FUNCTION_BLOCK fbEthercatStateMachine
VAR
	InputState AT%I*	:UINT;	
	WcState AT%I* :BOOL;
	InternalEtherCatState : st_EthercatState;
	
{attribute 'OPC.UA.DA' := '0'}	
	State :UINT;
		
{attribute 'OPC.UA.DA' := '0'}
	Error:UINT;
	
END_VAR

// table of states https://infosys.beckhoff.com/english.php?content=../content/1033/b110_ethercat_optioninterface/1984417163.html&id=
// uint is 16 bit final 4 bit are state first 12 are error 
State := InputState AND 16#000F;
Error := InputState AND 16#FFF0;
InternalEtherCatState.State:= UINT_TO_INT(State);
InternalEtherCatState.Error := UINT_TO_INT(Error);
InternalEtherCatState.DataInvalid := WcState;

METHOD FB_init : BOOL
VAR_INPUT
	bInitRetains : BOOL; // if TRUE, the retain variables are initialized (warm start / cold start)
	bInCopyCode : BOOL;  // if TRUE, the instance afterwards gets moved into the copy code (online change)
	EtherCatAddr : T_AmsNetID;
	nSlaveAddr : UINT;
END_VAR
InternalEtherCatState.nSlaveAddr:= nSlaveAddr;
InternalEtherCatState.EtherCatAddr := EtherCatAddr;
END_METHOD

METHOD GetState : BOOL
VAR_IN_OUT
	State : st_EthercatState;
END_VAR
State := InternalEtherCatState;
END_METHOD

END_FUNCTION_BLOCK

(* stored: Version 1.1.0.1, ProductVersion 3.1.4024.12
   POU fbEthercatStateMachine: Id {a8791b52-a045-4075-a09f-42bf13c3cfcd}, SpecialFunc None
   Method FB_init: Id {434a7edc-5ca9-4055-89dc-dc1a286dc610}
   Method GetState: Id {ce06c045-a69b-4b8e-a860-2028ae9368bf} *)
